TYPE ST_MyStruct :
STRUCT
    number      : LREAL;
    text        : STRING(10);
END_STRUCT
END_TYPE

(* stored: Version 1.1.0.1, ProductVersion 3.1.4024.11
   DUT ST_MyStruct: Id {111e5770-8d5b-4d8e-bf7d-bb6f31cde823} *)
